// Mitsubishi GX Works2 project: test2   PLC: Q03UDV

PROGRAM MAIN
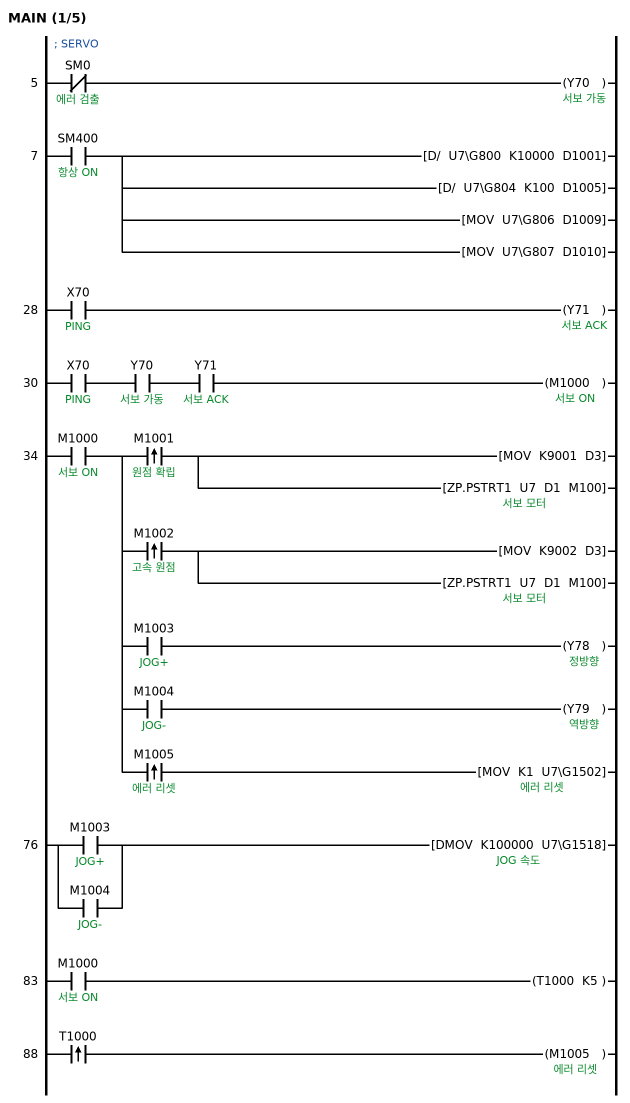
; SERVO
5     LDI     SM0  ; 에러 검출
      OUT     Y70  ; 서보 가동
7     LD      SM400  ; 항상 ON
      D/      U7\G800 K10000 D1001
      D/      U7\G804 K100 D1005
      MOV     U7\G806 D1009
      MOV     U7\G807 D1010
28    LD      X70  ; PING
      OUT     Y71  ; 서보 ACK
30    LD      X70  ; PING
      AND     Y70  ; 서보 가동
      AND     Y71  ; 서보 ACK
      OUT     M1000  ; 서보 ON
34    LD      M1000  ; 서보 ON
      MPS
      ANDP    M1001  ; 원점 확립
      MOV     K9001 D3
      ZP.PSTRT1 U7 D1 M100  ; 서보 모터
      MRD
      ANDP    M1002  ; 고속 원점
      MOV     K9002 D3
      ZP.PSTRT1 U7 D1 M100
      MRD
      AND     M1003  ; JOG+
      OUT     Y78  ; 정방향
      MRD
      AND     M1004  ; JOG-
      OUT     Y79  ; 역방향
      MPP
      ANDP    M1005  ; 에러 리셋
      MOV     K1 U7\G1502  ; 에러 리셋
76    LD      M1003  ; JOG+
      OR      M1004  ; JOG-
      DMOV    K100000 U7\G1518  ; JOG 속도
83    LD      M1000  ; 서보 ON
      OUT     T1000 K5
88    LDP     T1000
      OUT     M1005  ; 에러 리셋
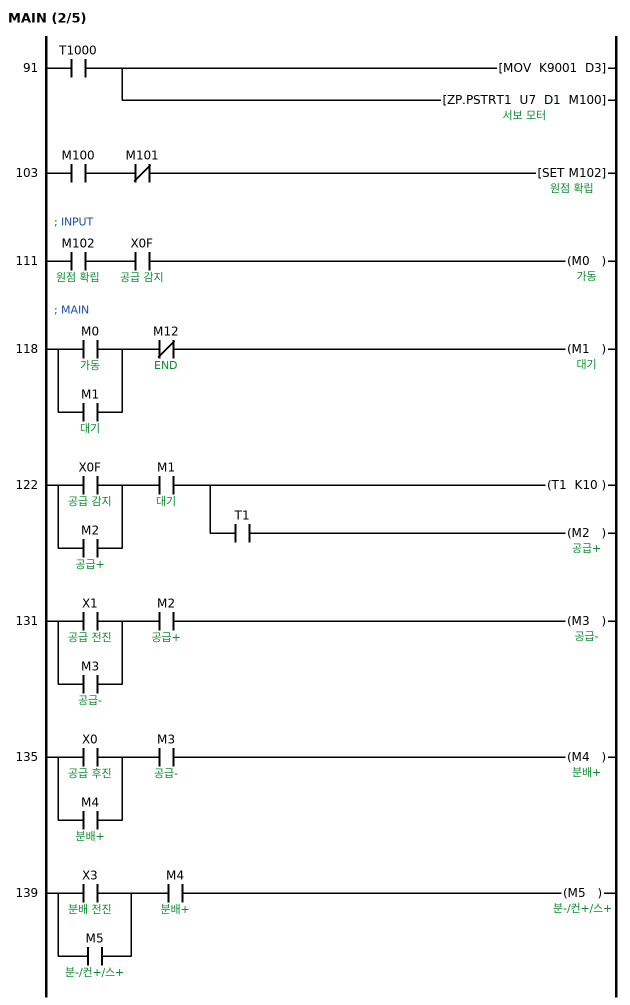
91    LD      T1000
      MOV     K9001 D3
      ZP.PSTRT1 U7 D1 M100
103   LD      M100
      ANI     M101
      SET     M102  ; 원점 확립
; INPUT
111   LD      M102  ; 원점 확립
      AND     X0F  ; 공급 감지
      OUT     M0  ; 가동
; MAIN
118   LD      M0  ; 가동
      OR      M1  ; 대기
      ANI     M12  ; END
      OUT     M1  ; 대기
122   LD      X0F  ; 공급 감지
      OR      M2  ; 공급+
      AND     M1  ; 대기
      OUT     T1 K10
      AND     T1
      OUT     M2  ; 공급+
131   LD      X1  ; 공급 전진
      OR      M3  ; 공급-
      AND     M2  ; 공급+
      OUT     M3  ; 공급-
135   LD      X0  ; 공급 후진
      OR      M4  ; 분배+
      AND     M3  ; 공급-
      OUT     M4  ; 분배+
139   LD      X3  ; 분배 전진
      OR      M5  ; 분-/컨+/스+
      AND     M4  ; 분배+
      OUT     M5  ; 분-/컨+/스+
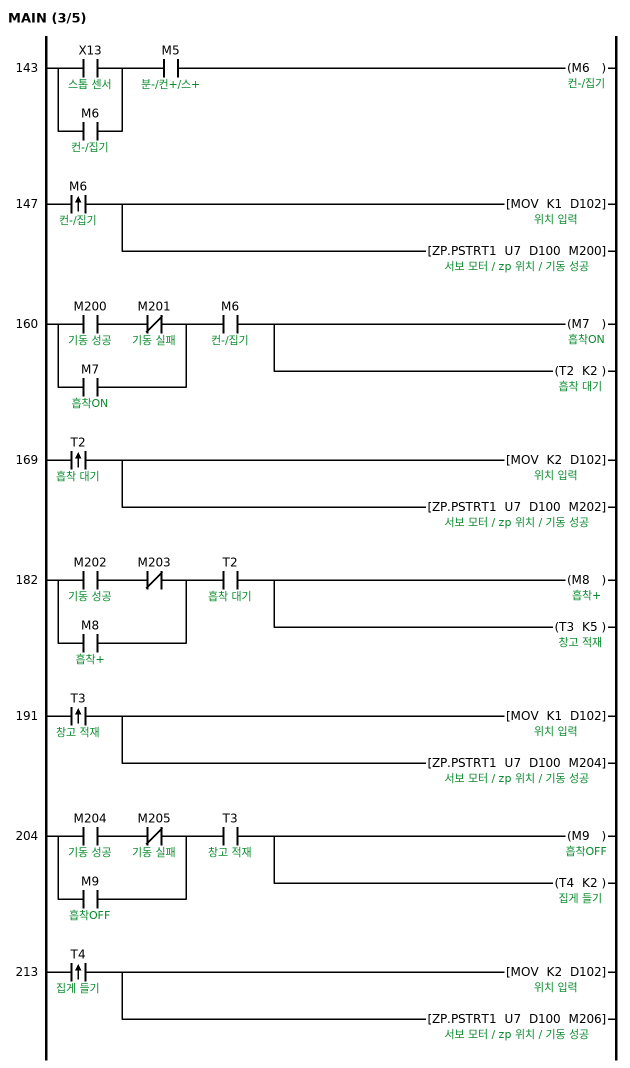
143   LD      X13  ; 스톱 센서
      OR      M6  ; 컨-/집기
      AND     M5  ; 분-/컨+/스+
      OUT     M6  ; 컨-/집기
147   LDP     M6  ; 컨-/집기
      MOV     K1 D102  ; 위치 입력
      ZP.PSTRT1 U7 D100 M200  ; zp 위치 / 기동 성공
160   LD      M200  ; 기동 성공
      ANI     M201  ; 기동 실패
      OR      M7  ; 흡착ON
      AND     M6  ; 컨-/집기
      OUT     M7  ; 흡착ON
      OUT     T2 K2  ; 흡착 대기
169   LDP     T2  ; 흡착 대기
      MOV     K2 D102
      ZP.PSTRT1 U7 D100 M202  ; 기동 성공
182   LD      M202  ; 기동 성공
      ANI     M203
      OR      M8  ; 흡착+
      AND     T2  ; 흡착 대기
      OUT     M8  ; 흡착+
      OUT     T3 K5  ; 창고 적재
191   LDP     T3  ; 창고 적재
      MOV     K1 D102
      ZP.PSTRT1 U7 D100 M204  ; 기동 성공
204   LD      M204  ; 기동 성공
      ANI     M205  ; 기동 실패
      OR      M9  ; 흡착OFF
      AND     T3  ; 창고 적재
      OUT     M9  ; 흡착OFF
      OUT     T4 K2  ; 집게 들기
213   LDP     T4  ; 집게 들기
      MOV     K2 D102
      ZP.PSTRT1 U7 D100 M206  ; 기동 성공
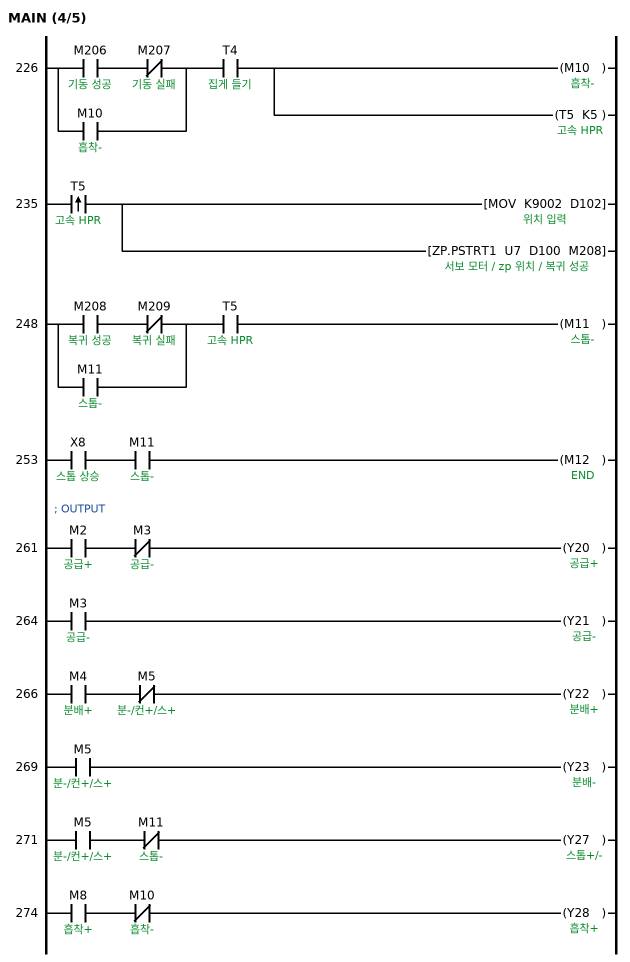
226   LD      M206  ; 기동 성공
      ANI     M207  ; 기동 실패
      OR      M10  ; 흡착-
      AND     T4  ; 집게 들기
      OUT     M10  ; 흡착-
      OUT     T5 K5  ; 고속 HPR
235   LDP     T5  ; 고속 HPR
      MOV     K9002 D102
      ZP.PSTRT1 U7 D100 M208  ; 복귀 성공
248   LD      M208  ; 복귀 성공
      ANI     M209  ; 복귀 실패
      OR      M11  ; 스톱-
      AND     T5  ; 고속 HPR
      OUT     M11  ; 스톱-
253   LD      X8  ; 스톱 상승
      AND     M11  ; 스톱-
      OUT     M12  ; END
; OUTPUT
261   LD      M2  ; 공급+
      ANI     M3  ; 공급-
      OUT     Y20  ; 공급+
264   LD      M3  ; 공급-
      OUT     Y21  ; 공급-
266   LD      M4  ; 분배+
      ANI     M5  ; 분-/컨+/스+
      OUT     Y22  ; 분배+
269   LD      M5  ; 분-/컨+/스+
      OUT     Y23  ; 분배-
271   LD      M5  ; 분-/컨+/스+
      ANI     M11  ; 스톱-
      OUT     Y27  ; 스톱+/-
274   LD      M8  ; 흡착+
      ANI     M10  ; 흡착-
      OUT     Y28  ; 흡착+
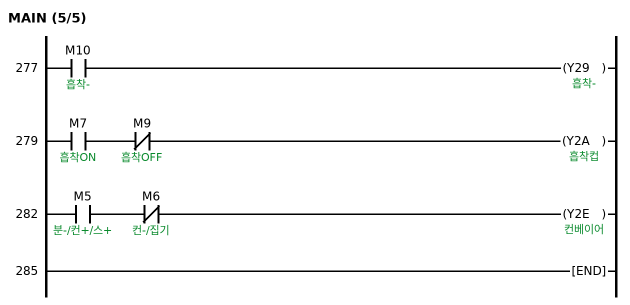
277   LD      M10  ; 흡착-
      OUT     Y29  ; 흡착-
279   LD      M7  ; 흡착ON
      ANI     M9  ; 흡착OFF
      OUT     Y2A  ; 흡착컵
282   LD      M5  ; 분-/컨+/스+
      ANI     M6  ; 컨-/집기
      OUT     Y2E  ; 컨베이어
285   END
END_PROGRAM

// device comments not shown above
X2  ; 분배 후진
X9  ; 스톱 하강
X0A  ; 흡착 후진
X0B  ; 흡착 전진
